// TwinCAT 3 PLC project PLCStudent
// ProgramVersion: 3.1.4026.20
// libraries:
//   Tc2_Standard, * (Beckhoff Automation GmbH)
//   Tc2_System, * (Beckhoff Automation GmbH)
//   Tc3_Module, * (Beckhoff Automation GmbH)
// project tree:
//   GVLs/ GVL.TcGVL
//   / PlcTask.TcTTO
//   POUs/ Control_FBD.TcPOU, MAIN.TcPOU
// (motion and I/O tree: see PLC project plcsim)
// real-time tasks:
//   TASK PlcTask: cycle T#20ms, priority 20, ADS port 350
// variable links:
//   PLCSim/PLCSim Instance <-> PLCStudent/PLCStudent Instance
//     PlcTask Inputs/GVL.iiDisplayElevat <-> PlcTask Outputs/GVL.qiDispElevat
//     PlcTask Inputs/GVL.ixDoorClose <-> PlcTask Outputs/GVL.qxDoorClose
//     PlcTask Inputs/GVL.ixLampElevat1 <-> PlcTask Outputs/GVL.qxLampElevat1
//     PlcTask Inputs/GVL.ixLampElevat2 <-> PlcTask Outputs/GVL.qxLampElevat2
//     PlcTask Inputs/GVL.ixLampElevat3 <-> PlcTask Outputs/GVL.qxLampElevat3
//     PlcTask Inputs/GVL.ixLampLevel1 <-> PlcTask Outputs/GVL.qxLampAtLevel1
//     PlcTask Inputs/GVL.ixLampLevel2 <-> PlcTask Outputs/GVL.qxLampAtLevel2
//     PlcTask Inputs/GVL.ixLampLevel3 <-> PlcTask Outputs/GVL.qxLampAtLevel3
//     PlcTask Inputs/GVL.ixMotorDown <-> PlcTask Outputs/GVL.qxMotorDown
//     PlcTask Inputs/GVL.ixMotorUp <-> PlcTask Outputs/GVL.qxMotorUp
//     PlcTask Outputs/GVL.qxButtElevat1 <-> PlcTask Inputs/GVL.ixButtInsideElevat1
//     PlcTask Outputs/GVL.qxButtElevat2 <-> PlcTask Inputs/GVL.ixButtInsideElevat2
//     PlcTask Outputs/GVL.qxButtElevat3 <-> PlcTask Inputs/GVL.ixButtInsideElevat3
//     PlcTask Outputs/GVL.qxButtGreen <-> PlcTask Inputs/GVL.ixButtGreen
//     PlcTask Outputs/GVL.qxButtLevel1 <-> PlcTask Inputs/GVL.ixButtonAtLevel1
//     PlcTask Outputs/GVL.qxButtLevel2 <-> PlcTask Inputs/GVL.ixButtonAtLevel2
//     PlcTask Outputs/GVL.qxButtLevel3 <-> PlcTask Inputs/GVL.ixButtonAtLevel3
//     PlcTask Outputs/GVL.qxButtRed <-> PlcTask Inputs/GVL.ixButtRed
//     PlcTask Outputs/GVL.qxDoorClosed <-> PlcTask Inputs/GVL.ixDoorClosed
//     PlcTask Outputs/GVL.qxDoorOpen <-> PlcTask Inputs/GVL.ixDoorOpen
//     PlcTask Outputs/GVL.qxElevatLevel1 <-> PlcTask Inputs/GVL.ixSensorAtLevel1
//     PlcTask Outputs/GVL.qxElevatLevel2 <-> PlcTask Inputs/GVL.ixSensorAtLevel2
//     PlcTask Outputs/GVL.qxElevatLevel3 <-> PlcTask Inputs/GVL.ixSensorAtLevel3

CONFIGURATION PLCStudent
    RESOURCE PLC ON TwinCAT3
        TASK PlcTask(INTERVAL := T#20ms, PRIORITY := 20);
        PROGRAM MAIN WITH PlcTask : MAIN;
    END_RESOURCE
END_CONFIGURATION

// ---- GVLs/GVL.TcGVL
{attribute 'qualified_only'}
VAR_GLOBAL
//Input to PLC from process
	ixButtonAtLevel1		AT %I*:	BOOL;		(* Button at level 1 *)
	ixButtonAtLevel2		AT %I*:	BOOL;		(* Button at level 2 *)
	ixButtonAtLevel3		AT %I*:	BOOL;		(* Button at level 3 *)

	ixSensorAtLevel1 		AT %I*: BOOL;		(* Sensor at level 1 for elevator presence *)
	ixSensorAtLevel2 		AT %I*: BOOL;		(* Sensor at level 2 for elevator presence *)
	ixSensorAtLevel3 		AT %I*: BOOL;		(* Sensor at level 3 for elevator presence *)

	ixButtGreen 			AT %I*:	BOOL;		(* Green button *)
	ixButtRed				AT %I*:	BOOL;		(* Red button, normally closed *)

	ixButtInsideElevat1		AT %I*:	BOOL;		(* Button 1 inside elevator PLCSim only *)
	ixButtInsideElevat2		AT %I*:	BOOL;		(* Button 2 inside elevator PLCSim only *)
	ixButtInsideElevat3		AT %I*:	BOOL;		(* Button 3 inside elevator PLCSim only *)
	
	ixDoorClosed			AT %I*: BOOL;		(* Sensor for door closed PLCSim only *)
	ixDoorOpen				AT %I*:	BOOL;		(* Sensor for door open   PLCSim only *)

//Output from PLC to process
	qxLampAtLevel1		AT %Q*:	BOOL;		(* Lamp at level 1*)
	qxLampAtLevel2		AT %Q*:	BOOL;		(* Lamp at level 2*)
	qxLampAtLevel3		AT %Q*:	BOOL;		(* Lamp at level 3*)
	
	qxMotorDown			AT %Q*:	BOOL;		(* Run motor down *)
	qxMotorUp			AT %Q*:	BOOL;		(* Run motor up *)

	qxLampElevat1 		AT %Q*:	BOOL;		(* Lamp 1 inside elevator PLCSim only*)
	qxLampElevat2 		AT %Q*:	BOOL;		(* Lamp 2 inside elevator PLCSim only *)
	qxLampElevat3 		AT %Q*:	BOOL;		(* Lamp 3 inside elevator PLCSim only *)

	qxDoorClose			AT %Q*:	BOOL;		(* Close door and keep it closed  PLCSim only *)
	qiDispElevat 		AT %Q*:	UINT;		(* Integer display inside elevator PLCSim only *)
	qxButtonAtLevel1: BOOL;
END_VAR

// ---- POUs/MAIN.TcPOU
PROGRAM MAIN
VAR
END_VAR

Control_FBD();

END_PROGRAM

// ---- POUs/Control_FBD.TcPOU
PROGRAM Control_FBD
VAR
END_VAR

END_PROGRAM
